// Mitsubishi GX Works2 project: GX W2 L4 Ex 1 DK C   PLC: FX3G

// global labels: Global1
VAR_GLOBAL
  iHallway_SW1 AT X001 : BOOL;
  iHallway_SW2 AT X002 : BOOL;
  oHallway_Light AT Y001 : BOOL;
  iStairs_SW1 AT X003 : BOOL;
  iStairs_SW2 AT X004 : BOOL;
  oStairs_Light AT Y002 : BOOL;
END_VAR

// task Task_01 (event TRUE, interval 0, priority 31): POU_01

PROGRAM POU_01
VAR
  Hallway_Control : fb_2_Way_SW;
  Stairs_Control : fb_2_Way_SW;
END_VAR
(* structured ladder/FBD written out as ST: instructions are called as NAME(EN, inputs, outputs); _pN, _eN, _tN stand for wires *)
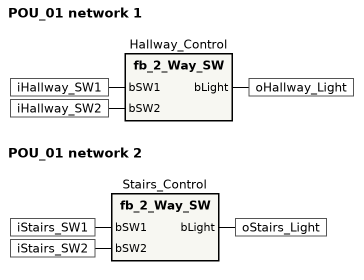
(* network 1 *)
Hallway_Control(bSW1 := iHallway_SW1, bSW2 := iHallway_SW2, bLight => oHallway_Light);
(* network 2 *)
Stairs_Control(bSW1 := iStairs_SW1, bSW2 := iStairs_SW2, bLight => oStairs_Light);
END_PROGRAM

FUNCTION_BLOCK fb_2_Way_SW
VAR_INPUT
  bSW1 : BOOL;
  bSW2 : BOOL;
END_VAR
VAR_OUTPUT
  bLight : BOOL;
END_VAR
(* structured ladder/FBD written out as ST: instructions are called as NAME(EN, inputs, outputs); _pN, _eN, _tN stand for wires *)
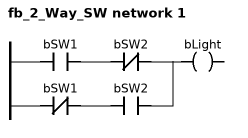
(* network 1 *)
bLight := (bSW1 AND NOT bSW2) OR (NOT bSW1 AND bSW2);
END_FUNCTION_BLOCK
